// TIA Portal V17 export
// export: Created 2024-08-26T21:07:17.7496416Z, ExportSetting WithDefaults, DisplayName Totally Integrated Automation Portal, DisplayVersion V17 Update 7, DisplayName TIA Portal Openness, DisplayVersion V17 Update 7, DisplayName TIA Portal Version Control Interface, DisplayVersion V17, DisplayName SINAMICS Startdrive Advanced, DisplayVersion V17 SP2, DisplayName SINAMICS Startdrive G110M, G120, G120C, G120D, G120P, G115D, DisplayVersion V17 SP2, DisplayName SINAMICS Startdrive G130, G150, S120, S150, SINAMICS MV, S210, DisplayVersion V17 SP2, DisplayName STEP 7 Professional, DisplayVersion V17 Update 7, DisplayName STEP 7 Safety, DisplayVersion V17 Update 6, DisplayName WinCC Advanced / Unified PC, DisplayVersion V17 Update 7
FUNCTION "FC_SD_TIMER" : Void   // FC401, LAD
TITLE = Standard simple SD timer
{ S7_Optimized_Access := 'FALSE' }
FAMILY : system
VERSION : 1.0
// stored: AutoNumber false, IsIECCheckEnabled false, SetENOAutomatically false, UDAEnableTagReadback false
   VAR_INPUT
      iPULSE : Bool;   // time impulse
      iENABLE : Bool;   // release of timer
      iTIMER_SET : Int;   // preset value
   END_VAR
   VAR_IN_OUT
      iqTIMER_STAT : Int;   // actual value
   END_VAR
   VAR_TEMP
      tOk : Bool;
   END_VAR
BEGIN

REGION Network 1: If not enabled, then reset actual value of timer
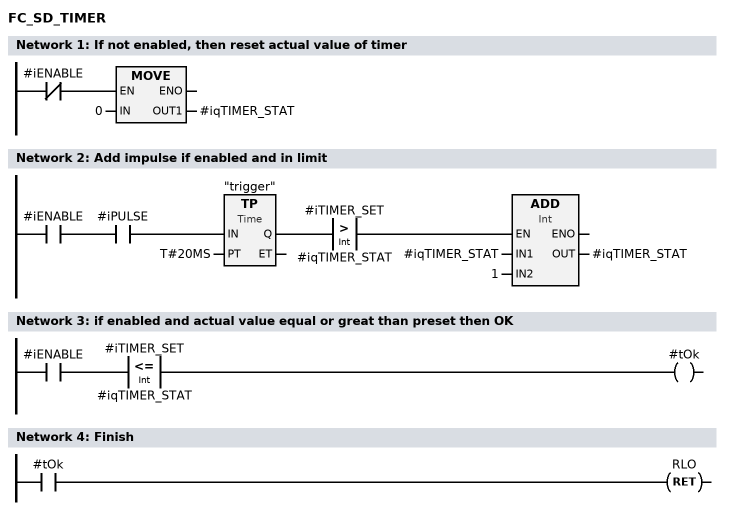
   RUNG wire#powerrail
      I_Contact( #iENABLE )
      { S7_GenerateENO := "TRUE" } Move(in := 0, out1 => #iqTIMER_STAT)
   END_RUNG
   // the same network as SCL:
   IF NOT #iENABLE THEN #iqTIMER_STAT := 0; END_IF;
END_REGION

REGION Network 2: Add impulse if enabled and in limit
   RUNG wire#powerrail
      Contact( #iENABLE )
      Contact( #iPULSE )
      { S7_Templates := "time_type := Time" } "trigger".TP(pt := T#20MS, et =>)
      { S7_Templates := "SrcType := Int" } GT_Contact(in1 := #iTIMER_SET, in2 := #iqTIMER_STAT)
      { S7_Templates := "SrcType := Int"; S7_GenerateENO := "TRUE" } Add(in1 := #iqTIMER_STAT, in2 := 1, out => #iqTIMER_STAT)
   END_RUNG
   // the same network as SCL:
   "trigger".TP(IN := #iENABLE AND #iPULSE, PT := T#20MS);
   IF "trigger".Q AND (#iTIMER_SET > #iqTIMER_STAT) THEN #iqTIMER_STAT := #iqTIMER_STAT + 1; END_IF;
END_REGION

REGION Network 3: if enabled and actual value equal or great than preset then OK
   RUNG wire#powerrail
      Contact( #iENABLE )
      { S7_Templates := "SrcType := Int" } LE_Contact(in1 := #iTIMER_SET, in2 := #iqTIMER_STAT)
      Coil( #tOk )
   END_RUNG
   // the same network as SCL:
   #tOk := #iENABLE AND (#iTIMER_SET <= #iqTIMER_STAT);
END_REGION

REGION Network 4: Finish
   IF #tOk THEN
       ENO := TRUE;
       RETURN;
   END_IF;
END_REGION
END_FUNCTION
